{attribute 'qualified_only'}
VAR_GLOBAL
END_VAR

(* stored: Version 1.1.0.1, ProductVersion 3.1.4022.7
   GVL GVL_03_Delay_Servo_Motor: Id {3c367ee2-9e52-4d8e-b0cb-d1707bb7a552} *)
